Staubli VAL3: default.pjx

--- default.pjx ---
Parameters version=s7.7.2 stackSize=5000 millimeterUnit=true
Program file=start.pgx
Program file=stop.pgx
Data file=default.dtx

--- default.dtx ---
mdesc mNomSpeed = {blend=joint, accel=100, vel=100, decel=100, tmax=99999, rmax=99999, leave=50, reach=50}

--- start.pgx ---
program start()
begin
end
